Universal Robots PolyScope program: PickAndPlace_App_Final.urp

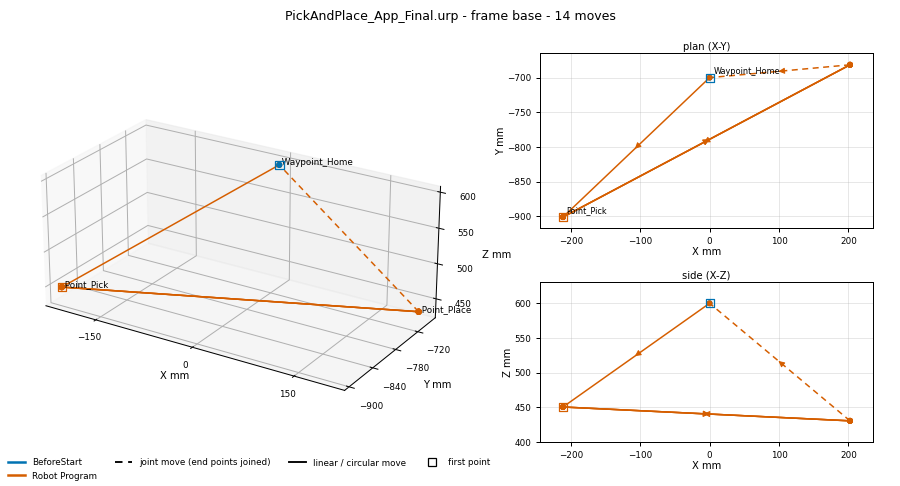
[picture p0: tool path of PickAndPlace_App_Final.urp in frame base, 14 of 20 moves have a stored position in this frame; points joined in program order, loops and branches not executed]
Program PickAndPlace_App_Final (installation=default directory=/home/ur/ursim-current/programs/new folder createdIn=5.11.4.108353 lastSavedIn=5.11.4.108353 robotSerialNumber=20195299999)
Calibrated DH parameters: a=[0, -0.6127, -0.57155, 0, 0, 0]; d=[0.1807, 0, 0, 0.17415, 0.11985, 0.11655]; alpha=[1.570796, 0, 0, 1.570796, -1.570796, 0]; deltaTheta=[0, 0, 0, 0, 0, 0]
BeforeStart
  v_count_of_obj := 3
  v_obj_height := 0.030
  v_actual_state := 1
  v_inv_mode := False
  v_counter := 0
  v_pick_offset := p[0.0,0.0,0.0,0.0,0.0,0.0]
  v_place_offset := p[0.0,0.0,0.0,0.0,0.0,0.0]
  v_pick_z := 0.2
  v_place_z := 0.2
  Script: Point_Place[2]=0.415+v_place_z
  Script: Point_Pick[2]=0.415+v_pick_z
  v_rpy_vec_pick := rotvec2rpy([Point_Pick[3],Point_Pick[4],Point_Pick[5]])
  v_rot_vec_pick := rpy2rotvec([3.142,0.0,v_rpy_vec_pick[2]])
  Script: Point_Pick[3]=v_rot_vec_pick[0]
  Script: Point_Pick[4]=v_rot_vec_pick[1]
  Script: Point_Pick[5]=v_rot_vec_pick[2]
  v_rpy_vec_place := rotvec2rpy([Point_Place[3],Point_Place[4],Point_Place[5]])
  v_rot_vec_place := rpy2rotvec([3.142,0.0,v_rpy_vec_place[2]])
  Script: Point_Place[3]=v_rot_vec_place[0]
  Script: Point_Place[4]=v_rot_vec_place[1]
  Script: Point_Place[5]=v_rot_vec_place[2]
  MoveJ speed 20 deg/s, acceleration 40 deg/s^2 (useActiveTCP=true) feature=Base
    Waypoint Waypoint_Home: TCP in base x=0 y=-700 z=600 mm, rx=0.0687 ry=3.1392 rz=0.0004 rad; joints [-75.586, -89.259, -98.465, -82.227, 89.79, 16.88] deg; TCP offset x=0 y=0 z=0 mm, rx=0 ry=0 rz=0 rad
Robot Program (runOnlyOnce=false)
  Switch expression=v_actual_state
    Case (caseValue=1)
      If v_inv_mode== True
        v_actual_state := 3
      Else 
        v_actual_state := 2
    Case (caseValue=2)
      If v_counter<v_count_of_obj
        MoveL speed 100 mm/s, acceleration 500 mm/s^2 (useActiveTCP=true) feature=Base
          Waypoint Point_Pick: TCP in base x=-211.196 y=-900.852 z=450.637 mm, rx=-0.6821 ry=3.0639 rz=0.011 rad; joints [-92.319, -113.668, -84.051, -72.669, 89.759, -27.519] deg
          v_pick_offset := pose_trans(Point_Pick, p[0.0,0.0,v_pick_z-((v_count_of_obj-(v_counter+1))*v_obj_height),0.0,0.0,0.0])
          Waypoint Waypoint (Variable): variable(name=v_pick_offset)
          Waypoint Point_Pick: TCP in base x=-211.196 y=-900.852 z=450.637 mm, rx=-0.6821 ry=3.0639 rz=0.011 rad; joints [-92.319, -113.668, -84.051, -72.669, 89.759, -27.519] deg
          Waypoint Point_Place: TCP in base x=202.305 y=-681.495 z=430.682 mm, rx=0.5199 ry=3.0972 rz=0.0362 rad; joints [-59.407, -95.102, -109.935, -65.9, 90.602, 49.53] deg
          v_place_offset := pose_trans(Point_Place, p[0.0,0.0,v_place_z-(v_counter*v_obj_height),0.0,0.0,0.0])
          Waypoint Waypoint (Variable): variable(name=v_place_offset)
          Waypoint Point_Place: TCP in base x=202.305 y=-681.495 z=430.682 mm, rx=0.5199 ry=3.0972 rz=0.0362 rad; joints [-59.407, -95.102, -109.935, -65.9, 90.602, 49.53] deg
          Script: v_counter=v_counter+1
      Else 
        MoveJ speed 20 deg/s, acceleration 40 deg/s^2 (useActiveTCP=true) feature=Base
          Waypoint Waypoint_Home: TCP in base x=0 y=-700 z=600 mm, rx=0.0687 ry=3.1392 rz=0.0004 rad; joints [-75.586, -89.259, -98.465, -82.227, 89.79, 16.88] deg; TCP offset x=0 y=0 z=0 mm, rx=0 ry=0 rz=0 rad
        Halt
    Case (caseValue=3)
      If v_counter<v_count_of_obj
        MoveL speed 100 mm/s, acceleration 500 mm/s^2 (useActiveTCP=true) feature=Base
          Waypoint Point_Pick: TCP in base x=-211.196 y=-900.852 z=450.637 mm, rx=-0.6821 ry=3.0639 rz=0.011 rad; joints [-92.319, -113.668, -84.051, -72.669, 89.759, -27.519] deg
          v_pick_offset := pose_trans(Point_Pick, p[0.0,0.0,v_pick_z-((v_count_of_obj-(v_counter+1))*v_obj_height),0.0,0.0,0.0])
          Waypoint Waypoint (Variable): variable=v_pick_offset
          Waypoint Point_Pick: TCP in base x=-211.196 y=-900.852 z=450.637 mm, rx=-0.6821 ry=3.0639 rz=0.011 rad; joints [-92.319, -113.668, -84.051, -72.669, 89.759, -27.519] deg
          Waypoint Point_Place: TCP in base x=202.305 y=-681.495 z=430.682 mm, rx=0.5199 ry=3.0972 rz=0.0362 rad; joints [-59.407, -95.102, -109.935, -65.9, 90.602, 49.53] deg
          v_place_offset := pose_trans(Point_Place, p[0.0,0.0,v_place_z-(v_counter*v_obj_height),0.0,0.0,0.0])
          Waypoint Waypoint (Variable): variable=v_place_offset
          Waypoint Point_Place: TCP in base x=202.305 y=-681.495 z=430.682 mm, rx=0.5199 ry=3.0972 rz=0.0362 rad; joints [-59.407, -95.102, -109.935, -65.9, 90.602, 49.53] deg
          Script: v_counter=v_counter+1
      Else 
        v_actual_state := 4
    Case (caseValue=4)
      If v_counter>0
        MoveL speed 100 mm/s, acceleration 500 mm/s^2 (useActiveTCP=true) feature=Base
          Waypoint Point_Place: TCP in base x=202.305 y=-681.495 z=430.682 mm, rx=0.5199 ry=3.0972 rz=0.0362 rad; joints [-59.407, -95.102, -109.935, -65.9, 90.602, 49.53] deg
          v_pick_offset := pose_trans(Point_Place, p[0.0,0.0,v_place_z-((v_counter-1)*v_obj_height),0.0,0.0,0.0])
          Waypoint Waypoint (Variable): variable=v_pick_offset
          Waypoint Point_Place: TCP in base x=202.305 y=-681.495 z=430.682 mm, rx=0.5199 ry=3.0972 rz=0.0362 rad; joints [-59.407, -95.102, -109.935, -65.9, 90.602, 49.53] deg
          Waypoint Point_Pick: TCP in base x=-211.196 y=-900.852 z=450.637 mm, rx=-0.6821 ry=3.0639 rz=0.011 rad; joints [-92.319, -113.668, -84.051, -72.669, 89.759, -27.519] deg
          v_place_offset := pose_trans(Point_Pick, p[0.0,0.0,v_pick_z-((v_count_of_obj-v_counter)*v_obj_height),0.0,0.0,0.0])
          Waypoint Waypoint (Variable): variable=v_place_offset
          Waypoint Point_Pick: TCP in base x=-211.196 y=-900.852 z=450.637 mm, rx=-0.6821 ry=3.0639 rz=0.011 rad; joints [-92.319, -113.668, -84.051, -72.669, 89.759, -27.519] deg
          Script: v_counter=v_counter-1
      Else 
        v_actual_state := 3
